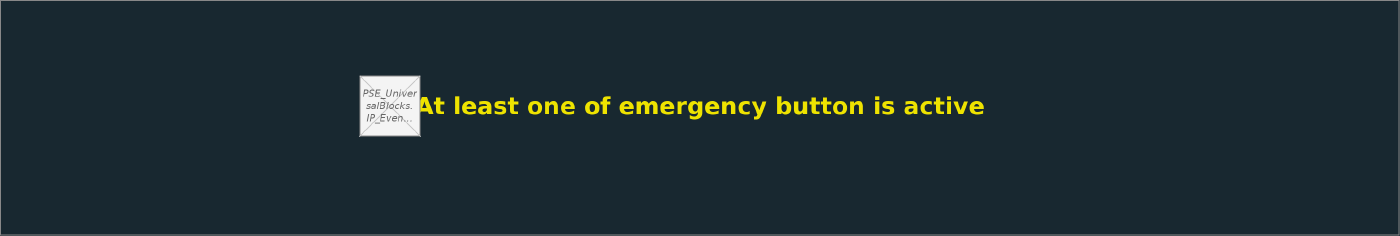
VISUALIZATION InitializingEStopActive  // 1480x250
    Label (0,92 1480x40), "At least one of emergency button is active"
    Image (380,80 64x64), image: PSE_UniversalBlocks.IP_EventSeverity.error
END_VISUALIZATION

(* stored: Version 1.1.0.1, ProductVersion 3.1.4024.9
   Visu InitializingEStopActive: Id {48d285ad-28f6-4a20-a88b-63b227764215} *)
